// Mitsubishi GX Works2 project: questão_6   PLC: Q03UDV
// LRI_2023

PROGRAM MAIN
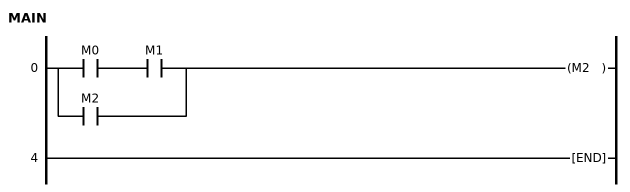
0     LD      M0
      AND     M1
      OR      M2
      OUT     M2
4     END
END_PROGRAM
